// TIA Portal V17 export
// export: Created 2025-03-07T09:24:40.9897052Z, ExportSetting WithDefaults, DisplayName Totally Integrated Automation Portal, DisplayVersion V17 Update 8, DisplayName TIA Portal Openness, DisplayVersion V17 Update 8, DisplayName TIA Portal Version Control Interface, DisplayVersion V17, DisplayName SINAMICS Startdrive Advanced, DisplayVersion V17 SP2, DisplayName SINAMICS Startdrive G110M, G120, G120C, G120D, G120P, G115D, DisplayVersion V17 SP2, DisplayName SINAMICS Startdrive G130, G150, S120, S150, SINAMICS MV, S210, DisplayVersion V17 SP2, DisplayName STEP 7 Professional, DisplayVersion V17 Update 8, DisplayName SINUMERIK ONE STEP 7 Toolbox, DisplayVersion V17 Update 12, DisplayName SINUMERIK 840D sl STEP 7 Toolbox, DisplayVersion V17 Update 12, DisplayName STEP 7 Safety, DisplayVersion V17 Update 6, DisplayName WinCC Advanced, DisplayVersion V17 Update 8
TYPE "CYCLES"
// stored: IsFailsafeCompliant false
   STRUCT
      GENERAL_CONDITIONS : Bool;   // CHANGE GENERAL CONDITIONS / CHANGE CYCLE GENERAL CONDITIONS
      INITIAL_CONDITIONS : Bool;   // CHANGE INITIAL CONDITIONS / CHANGE CYCLE INITIAL CONDITIONS
      ENABLE_REQUEST : Bool;   // ENABLE REQUEST
      DISABLE_REQUEST : Bool;   // DISABLE REQUEST
      TOGGLE_COMMAND_P : Bool;   // TOGGLE COMAND PULSE / TOGGLE COMMAND PULSE
      WARNING_GONE : Bool;   // TOGGLE COMMAND AUXILIARY / WARNING GONE
      GENERAL_CONDITIONS_HELP : Bool;   // GENERAL CONDITIONS HELP / CHANGE CYCLE GENERAL CONDITIONS HELP
      INITIAL_CONDITIONS_HELP : Bool;   // INITIAL CONDITIONS HELP / CHANGE CYCLE INITIAL CONDITIONS HELP
      CYCLE_SELECTED : Bool;   // MODE SELECTED / CYCLE SELECTED
      CYCLE_SELECTED_AUX : Bool;   // AUXILIARY MODE SELECTED / CYCLE SELECTED AUXILIARY
      CYCLE_COMPLETED : Bool;   // COMPLETED / CYCLE COMPLETED
      MACHINE_EMPTY : Bool;   // MACHINE EMPTY
      MACHINE_EMPTY_MANUAL_LOAD_SELECTED : Bool;   // MACHINE EMPTY WITH MANUAL LOAD SELECTED / MACHINE EMPTY MANUAL LOAD SELECTED
      MACHINE_EMPTY_WO_MANUAL_LOAD_SELECTED : Bool;   // MACHINE EMPTY WITHOUT MANUAL LOAD SELECTED
      RESET_FULL_DEPTH_DRY_CYCLE_DISABLED : Bool;   // RESET DEPTHS WHEN DRY CYCLE DISABLED / RESET FULL DEPTH DRY CYCLE DISABLED
      RESET_FULL_DEPTHS_AUX : Bool;   // RESET FULL DEPTHS AUXILIARY
      CYCLE_SEOC : Bool;   // CYCLE STOP END OF CYCLE
      CYCLE_IS : Bool;   // CYCLE IMMEDIATE STOP
   END_STRUCT;
END_TYPE
